TYPE ST_ControlComau :
STRUCT
	u : ARRAY[0..5] OF LREAL;

END_STRUCT
END_TYPE

(* stored: Version 1.1.0.1, ProductVersion 3.1.4026.8
   DUT ST_ControlComau: Id {73075925-8e60-4fe6-994b-5a1e70361c0b} *)
